{attribute 'GeneratedUsingTerminal: EK1122-0000-0018'}
{attribute addProperty BoxType "EK1122-0000-0018"}
{attribute addProperty Id "Beckhoff_ELM37xxsub_EK1100EK1100_1FC0878B2"}
{attribute addProperty CRC "3826114437"}
{attribute addProperty Size "2"}
TYPE Beckhoff_ELM37xxEK1122_E40DDF85 EXTENDS EK1122_1FC0878B :
STRUCT
	{attribute addProperty Name "Beckhoff_ELM37xxsub_EK1100"}
	{attribute addProperty PreviousPort "Beckhoff ELM37xxEK1122 : D"}
	Beckhoff_ELM37xxsub_EK1100 : EK1100_1FC0878B;
END_STRUCT
END_TYPE

(* stored: Version 1.2.0.0, ProductVersion 3.1.4024.9
   DUT Beckhoff_ELM37xxEK1122_E40DDF85: Id {46d00438-7e84-40a2-885e-7f7243e20269} *)
